// TIA Portal V20 export
DATA_BLOCK "Instance_FB_Digital_Outputs_DB"   // DB103
// stored: AutoNumber false, InstanceOfName FB_Digital_Outputs, InstanceOfType FB
"FB_Digital_Outputs"
   // VAR_INPUT
   //    DB_Blink_Button_Light : Bool;
   //    DB_Turn_On_Button_Light : Bool;
   //    DB_Light_Fail_Test : Bool;
   //    DB_Light_Approve_Test : Bool;
   //    DB_Digital_Output_3 : Bool;
   //    Clock_1Hz : Bool;
   // END_VAR
   // VAR_OUTPUT
   //    Q_Button_Light : Bool;
   //    Q_Light_Fail_Test : Bool;
   //    Q_Light_Approve_Test : Bool;
   //    Q_Digital_Output_3 : Bool;
   // END_VAR
   // VAR
   //    Timer_Delay_Fail_Test { S7_SetPoint := 'True'} : TON_TIME;
   //    Timer_Delay_Approve_Test { S7_SetPoint := 'True'} : TON_TIME;
   // END_VAR
BEGIN
END_DATA_BLOCK
